	    REGION STATE MACHINE STEPS
	      CASE #statState OF
	        0://STATE 0
	          #statDriveControl.xDriveEnable := #statEnabled;
	          #statDriveControl.xDriveRun := FALSE;
	          #statDriveControl.xDriveEmergencyStop := #statSafetyIsOk;
	          #statDriveControl.iDriveSpeedRef_percent := 0.0;
	          #statBrushingIsDone := false;
	          #statBrushDriveControl.xDriveEnable := #statEnabled;
	          #statBrushDriveControl.xDriveRun := FALSE;
	          #statBrushDriveControl.xDriveEmergencyStop := #statSafetyIsOk;
	          #statBrushDriveControl.iDriveSpeedRef_percent := 0.0;
	          #statBrushing := false;
	          #statTrayStopperExtend := FALSE;
	          #statBrushingIsDoneLock := FALSE;

	        1://STATE 1
	          #statDriveControl.xDriveEnable := #statEnabled;
	          #statDriveControl.xDriveRun := TRUE;
	          #statDriveControl.xDriveEmergencyStop := #statSafetyIsOk;
	          #statDriveControl.iDriveSpeedRef_percent := #statSpeed_percent;
	          #statBrushing := FALSE;
	          #statBrushDriveControl.xDriveEnable := #statEnabled;
	          #statBrushDriveControl.xDriveEmergencyStop := #statSafetyIsOk;
	          #statBrushDriveControl.xDriveRun := FALSE;

	        2://STATE 2
	          #statDriveControl.xDriveEnable := #statEnabled;
	          #statDriveControl.xDriveRun := FALSE;
	          #statDriveControl.xDriveEmergencyStop := #statSafetyIsOk;
	          #statDriveControl.iDriveSpeedRef_percent := 0.0;
	          #statTrayStopperExtend := FALSE;
	        3://STATE 3
	          #statDriveControl.xDriveEnable := false;
	          #statDriveControl.xDriveRun := FALSE;
	          #statDriveControl.xDriveEmergencyStop := #statSafetyIsOk;
	          #statDriveControl.iDriveSpeedRef_percent := 0.0;
	          #statBrushing := FALSE;
	          #statTrayStopperExtend := FALSE;
	          #statBrushDriveControl.xDriveRun := FALSE;
	        4://STATE 4
	          #statDriveControl.xDriveEnable := #statEnabled;
	          #statDriveControl.xDriveRun := FALSE;
	          #statDriveControl.xDriveEmergencyStop := false;
	          #statDriveControl.iDriveSpeedRef_percent := 0.0;
	          #statBrushing := FALSE;
	          #statTrayStopperExtend := FALSE;
	          #statDriveControl.xDriveEmergencyStop := FALSE;
	        5://STATE 5
	          #statDriveControl.xDriveEnable := #statEnabled;
	          #statDriveControl.xDriveRun := FALSE;
	          #statDriveControl.xDriveEmergencyStop := #statSafetyIsOk;
	          #statDriveControl.iDriveSpeedRef_percent := 0.0;
	          #statBrushDriveControl.xDriveEnable := #statEnabled;
	          #statBrushDriveControl.xDriveRun := TRUE;
	          #statBrushDriveControl.xDriveEmergencyStop := #statSafetyIsOk;
	          #statBrushDriveControl.iDriveSpeedRef_percent := #ConveyorInterface.commands.rBrushSpeed_percent;
	          #statBrushing := TRUE;
	        6://STATE 6
	          #statDriveControl.xDriveEnable := #statEnabled;
	          #statDriveControl.xDriveRun := #statRunConvInMaintenance;
	          #statDriveControl.xDriveEmergencyStop := #statSafetyIsOk;
	          #statDriveControl.iDriveSpeedRef_percent := #statSpeedInMaintenance_percent;
	          #statBrushDriveControl.xDriveEnable := #statEnabled;
	          #statBrushDriveControl.xDriveRun := #statRunBrushInMaintenance;
	          #statBrushDriveControl.xDriveEmergencyStop := #statSafetyIsOk;
	          #statBrushDriveControl.iDriveSpeedRef_percent := #statBrushSpeed_percent;
	          #statBrushing := #statBrushExtendInMaintenance;
	          #statTrayStopperExtend := #statTrayStopperExtendInMaintenance;
	        ELSE
	          #statDriveControl.xDriveEnable := false;
	          #statDriveControl.xDriveRun := FALSE;
	          #statDriveControl.xDriveEmergencyStop := #statSafetyIsOk;
	          #statDriveControl.iDriveSpeedRef_percent := 0.0;
	          #statBrushing := false;
	          #statBrushDriveControl.xDriveEnable := false;
	          #statBrushDriveControl.xDriveRun := FALSE;
	          #statBrushDriveControl.xDriveEmergencyStop := #statSafetyIsOk;
	          #statBrushDriveControl.iDriveSpeedRef_percent := 0.0;

	      END_CASE;
	    END_REGION STATE MACHINE STEPS

	  END_REGION STATE MACHINE

	  REGION POST-STATE MACHINE OPERATIONS
	    //operations in this block will be implemented in each cycle, disregarding the state

	  END_REGION POST-STATE MACHINE OPERATONS

	END_REGION LOGIC

	REGION WRITE OUTPUTS, CALL SUBFUNCTIONS
	  //drive control
	  #instConveyorDrive(driveControl := #statDriveControl,
	                     inPI4 := #ConveyorInterface.inputs.i_ConveyorSEWdrivePI4,
	                     driveStatus => #statDriveStatus,
	                     outPO4 => #ConveyorInterface.outputs.q_ConveyorSEWdrivePO4);

	  #ConveyorInterface.status.xFault := #statDriveStatus.xDriveFault;
	  #ConveyorInterface.status.wFaultCode.%X0 := #statDriveStatus.xDriveFault;
	  #ConveyorInterface.status.iStatus := #statState;

	  //brush drive control
	  #instBrushDrive(driveControl:=#statBrushDriveControl,
	                  inPI4:=#ConveyorInterface.inputs.i_BrushDrivePI4,
	                  driveStatus=>#statBrushDriveStatus,
	                  outPO4=>#ConveyorInterface.outputs.q_BrushDrivePO4);

	  #ConveyorInterface.status.xFault := #ConveyorInterface.status.xFault OR #statBrushDriveStatus.xDriveFault;
	  #ConveyorInterface.status.wFaultCode.%X1 := #statBrushDriveStatus.xDriveFault;

	  //brush control
	  #ConveyorInterface.outputs.q_xBrushExtend := #statBrushing;
	  //stopper control
	  #ConveyorInterface.outputs.q_xTrayStopperExtend := #statTrayStopperExtend;

	END_REGION WRITE OUTPUTS, CALL SUBFUNCTIONS
END_FUNCTION_BLOCK

FUNCTION_BLOCK "ClassConveyorWithEjectSEW"
{ S7_Optimized_Access := 'TRUE' }
VERSION : 0.3
   VAR_IN_OUT
      ConveyorInterface : "typeConveyorWithEjectInterface";
   END_VAR

   VAR
      statEnabled { ExternalAccessible := 'False'; ExternalVisible := 'False'; ExternalWritable := 'False'} : Bool;
      instTimeDelay {InstructionName := 'TON_TIME'; LibVersion := '1.0'; ExternalAccessible := 'False'; ExternalVisible := 'False'; ExternalWritable := 'False'; S7_SetPoint := 'False'} : TON_TIME;
      statState { ExternalAccessible := 'False'; ExternalVisible := 'False'; ExternalWritable := 'False'} : USInt;   // State Machine Step number
      statNumberOfStates { ExternalAccessible := 'False'; ExternalVisible := 'False'; ExternalWritable := 'False'} : USInt := 1;   // State Machine Number of Steps
      statReadyForState { ExternalAccessible := 'False'; ExternalVisible := 'False'; ExternalWritable := 'False'} : Array[0..9] of Bool;
      statCycleCounter { ExternalAccessible := 'False'; ExternalVisible := 'False'; ExternalWritable := 'False'} : USInt;   // class specific variables
      statStart { ExternalAccessible := 'False'; ExternalVisible := 'False'; ExternalWritable := 'False'} : Bool;
      statStop { ExternalAccessible := 'False'; ExternalVisible := 'False'; ExternalWritable := 'False'} : Bool;
      statFull { ExternalAccessible := 'False'; ExternalVisible := 'False'; ExternalWritable := 'False'} : Bool;
      statSafetyIsOk { ExternalAccessible := 'False'; ExternalVisible := 'False'; ExternalWritable := 'False'} : Bool;
      statReset { ExternalAccessible := 'False'; ExternalVisible := 'False'; ExternalWritable := 'False'} : Bool;
      statMaintenance { ExternalAccessible := 'False'; ExternalVisible := 'False'; ExternalWritable := 'False'} : Bool;
      statRunConvInMaintenance { ExternalAccessible := 'False'; ExternalVisible := 'False'; ExternalWritable := 'False'} : Bool;
      statExtendEjectInMaintenance { ExternalAccessible := 'False'; ExternalVisible := 'False'; ExternalWritable := 'False'} : Bool;
      statSpeed_percent { ExternalAccessible := 'False'; ExternalVisible := 'False'; ExternalWritable := 'False'} : Real;
      statSpeedInMaintenance_percent { ExternalAccessible := 'False'; ExternalVisible := 'False'; ExternalWritable := 'False'} : Real;
      statStartOffTrigger { ExternalAccessible := 'False'; ExternalVisible := 'False'; ExternalWritable := 'False'} : Bool;
      statStopOnTrigger { ExternalAccessible := 'False'; ExternalVisible := 'False'; ExternalWritable := 'False'} : Bool;
      statFullOnTrigger { ExternalAccessible := 'False'; ExternalVisible := 'False'; ExternalWritable := 'False'} : Bool;
      statVFDfault { ExternalAccessible := 'False'; ExternalVisible := 'False'; ExternalWritable := 'False'} : Bool;
      statTrayEjected { ExternalAccessible := 'False'; ExternalVisible := 'False'; ExternalWritable := 'False'} : Bool;
      statDriveControl { ExternalAccessible := 'False'; ExternalVisible := 'False'; ExternalWritable := 'False'} : "typeDriveControl";
      statDriveStatus { ExternalAccessible := 'False'; ExternalVisible := 'False'; ExternalWritable := 'False'} : "typeDriveStatus";   // instances
      instConveyorStartOffDelay {InstructionName := 'TOF_TIME'; LibVersion := '1.0'; ExternalAccessible := 'False'; ExternalVisible := 'False'; ExternalWritable := 'False'; S7_SetPoint := 'False'} : TOF_TIME;
      instConveyorStopOnDelay {InstructionName := 'TON_TIME'; LibVersion := '1.0'; ExternalAccessible := 'False'; ExternalVisible := 'False'; ExternalWritable := 'False'; S7_SetPoint := 'False'} : TON_TIME;
      instConveyorFullOnDelay {InstructionName := 'TON_TIME'; LibVersion := '1.0'; ExternalAccessible := 'False'; ExternalVisible := 'False'; ExternalWritable := 'False'; S7_SetPoint := 'False'} : TON_TIME;
      instEjectDelay {InstructionName := 'TON_TIME'; LibVersion := '1.0'; ExternalAccessible := 'False'; ExternalVisible := 'False'; ExternalWritable := 'False'; S7_SetPoint := 'False'} : TON_TIME;
      instConveyorDrive { ExternalAccessible := 'False'; ExternalVisible := 'False'; ExternalWritable := 'False'; S7_SetPoint := 'False'} : "classDriveSEW";
   END_VAR

   VAR CONSTANT
      NUMBER_OF_STATES_IN_STATE_MACHINE : USInt := 7;   // 0-Conveyor stopped, 1-Conveyor running, 2-Conveyor full, 3-Conveyor fault, 4-Conveyor estopped, 5-Conveyor ejecting, 6-maintenance mode
   END_VAR


BEGIN
	REGION BLOCK INFO HEADER
	  //===============================================================================
	  // OTOMAKEIT SOLUTIONS / (c)Copyright 2024
	  //-------------------------------------------------------------------------------
	  // Title:            ClassConveyorWithEjectSEW
	  // Comment/Function: Conveyor class for TIA Portal, using SEW VFD drive. The only
	  //                   difference from the standard conveyor is the addition of the
	  //       eject cylinder control at the end of the conveyor
	  // Parental class:   classConveyor
	  // Library/Family:   LOMS (Library OtoMakeit Solutions)
	  // Author:           Yuriy Mosiyenko, Otomakeit Solutions
	  // Tested with:
	  // Engineering:      TIA Portal V17
	  // Restrictions:
	  // Requirements:     PLC (S7-1200 / S7-1500)
	  //-------------------------------------------------------------------------------
	  // Change log table:
	  //             | Date       | Expert in charge       | Changes applied
	  //-------------|------------|------------------------|------------------------------
	  // Created     | 2024-08-27 | Yuriy Mosiyenko        | Created
	  // Last update | 2024-08-29 | Yuriy Mosiyenko        | Corrections
	  //===============================================================================
	  //Update comments:
	  //-------------------------------------------------------------------------------
	  //2024-08-27 - Created the class
	  //2024-08-29 - Maintenance mode added
	  //===============================================================================
	  //===============================================================================
	END_REGION

	REGION INIT
	  #statNumberOfStates := #NUMBER_OF_STATES_IN_STATE_MACHINE;
	  FOR #statCycleCounter := 0 TO #statNumberOfStates DO
	    #statReadyForState[#statCycleCounter] := FALSE;
	  END_FOR;

	END_REGION INIT

	REGION READ INPUTS
	  #statEnabled := #ConveyorInterface.commands.xEnable;
	  #statStart := #ConveyorInterface.commands.xStart;
	  #statStop := #ConveyorInterface.commands.xStop;
	  #statFull := #ConveyorInterface.commands.xConveyorFullStatus;
	  #statReset := #ConveyorInterface.commands.xReset;
	  #statMaintenance := #ConveyorInterface.commands.xMaintenance;
	  #statRunConvInMaintenance := #ConveyorInterface.commands.xRunConvInMaintenance;
	  #statExtendEjectInMaintenance := #ConveyorInterface.commands.xExtendEjectInMaintenance;
	  #statSpeed_percent := #ConveyorInterface.commands.rConveyorSpeed_percent;
	  #statSpeedInMaintenance_percent := #ConveyorInterface.commands.rConveyorSpeedInMaintenance_percent;
	  #statSafetyIsOk := #ConveyorInterface.commands.xSafetyIsOk;

	END_REGION READ INPUTS

	REGION LOGIC

	  REGION PRE-STATE MACHINE OPERATIONS
	    //operations in this block will be implemented in each cycle, disregarding the state
	    //
	    //If reset received, reset faults, and set state machine to initial state
	    IF #statReset THEN
	      #ConveyorInterface.status.xFault := FALSE;
	      #ConveyorInterface.status.wFaultCode := 0;
	      #statState := 0;
	    END_IF;
	    IF NOT #statEnabled THEN //if the conveyor is disabled, stop it and set the status to 0 (stopped and ready)
	      #ConveyorInterface.status.iStatus := 0;
	      #statState := 0;
	      #statStart := FALSE;
	      #statStop := FALSE;
	    END_IF;
	    //start off delay
	    #instConveyorStartOffDelay(IN := #statStart,
	                               PT := #ConveyorInterface.commands.tStartOffDelay,
	                               Q => #statStartOffTrigger);
	    //STOP off delay
	    #instConveyorStopOnDelay(IN := #statStop,
	                              PT := #ConveyorInterface.commands.tStopOnDelay,
	                              Q => #statStopOnTrigger);
	    //FULL off delay
	    #instConveyorFullOnDelay(IN := #statFull,
	                              PT := #ConveyorInterface.commands.tFullOnDelay,
	                              Q => #statFullOnTrigger);
	    //Eject delay and output control
	    #instEjectDelay(IN := #statState = 5,
	                    PT := #ConveyorInterface.commands.tEjectTime,
	                    Q => #statTrayEjected);

	  END_REGION PRE-STATE MACHINE OPERATONS

	  REGION STATE MACHINE
	    REGION STATE MACHINE CONTROL
	      //set the conditions for each state
	      //state 0 - stopped and ready, state 1 - running, state 2 - stopped and full, state 3 - faulty, state 4 - estopped, state 5 - tray ejecting, state 6 - maintenance mode

	      //state 0 - if conveyor was full and the full status is removed or conveyor was running and the start or stop command is removed or fault was removed or safety was restored
	      //keep in mind that the stop command is active if false
	      #statReadyForState[0] := (#statState = 2 AND NOT #statFull)
	      OR (#statState = 4 AND #statSafetyIsOk)
	      OR (#statState = 3 AND NOT #statVFDfault)
	      OR (#statState = 5 AND #statTrayEjected)
	      OR (#statState = 6 AND NOT #statMaintenance);

	      //state 1 - if the conveyor is not full and the safety is ok and the start command is active
	      #statReadyForState[1] := (#statState = 0 AND #statStart AND #statSafetyIsOk);

	      //state 2 - if the conveyor is full
	      #statReadyForState[2] := (#statState < 3 AND #statFullOnTrigger AND #statSafetyIsOk);

	      //state 3 - if the VFD fault is detected
	      #statReadyForState[3] := (#statState = 1 AND #statVFDfault);

	      //state 4 - if the safety is not ok
	      #statReadyForState[4] := NOT #statSafetyIsOk;

	      //state 5 - if the stop command is active and delay is over
	      #statReadyForState[5] := (#statState = 1 AND #statStopOnTrigger AND #statSafetyIsOk);

	      //state 6 - if the maintenance mode is active
	      #statReadyForState[6] := (#statState = 0 AND #statMaintenance);

	      //change state if condition is TRUE
	      FOR #statCycleCounter := 0 TO #statNumberOfStates - 1 DO
	        IF #statReadyForState[#statCycleCounter] THEN
	          #statState := #statCycleCounter;
	        END_IF;
	      END_FOR;

	      //do not go over the set number of steps
	      IF #statState >= #statNumberOfStates THEN
	        #statState := 0;
	      END_IF;

	    END_REGION STATE MACHINE CONTROL

	    REGION STATE MACHINE STEPS
	      CASE #statState OF
	        0://STATE 0 - stopped and ready
	          #statDriveControl.xDriveEnable := #statEnabled;
	          #statDriveControl.xDriveRun := FALSE;
	          #statDriveControl.xDriveEmergencyStop := #statSafetyIsOk;
	          #statDriveControl.iDriveSpeedRef_percent := 0.0;
	          #statTrayEjected := FALSE;
	        1://STATE 1 - running
	          #statDriveControl.xDriveEnable := #statEnabled;
	          #statDriveControl.xDriveRun := TRUE;
	          #statDriveControl.xDriveEmergencyStop := #statSafetyIsOk;
	          #statDriveControl.iDriveSpeedRef_percent := #statSpeed_percent;
	        2://STATE 2 - stopped and full
	          #statDriveControl.xDriveEnable := #statEnabled;
	          #statDriveControl.xDriveRun := FALSE;
	          #statDriveControl.xDriveEmergencyStop := #statSafetyIsOk;
	          #statDriveControl.iDriveSpeedRef_percent := 0.0;
	        3://STATE 3 - faulty
	          #statDriveControl.xDriveEnable := false;
	          #statDriveControl.xDriveRun := FALSE;
	          #statDriveControl.xDriveEmergencyStop := #statSafetyIsOk;
	          #statDriveControl.iDriveSpeedRef_percent := 0.0;
	        4://STATE 4 - estopped
	          #statDriveControl.xDriveEnable := #statEnabled;
	          #statDriveControl.xDriveRun := FALSE;
	          #statDriveControl.xDriveEmergencyStop := false;
	          #statDriveControl.iDriveSpeedRef_percent := 0.0;
	        5://STATE 5 - tray ejecting
	          #statDriveControl.xDriveEnable := #statEnabled;
	          #statDriveControl.xDriveRun := FALSE;
	          #statDriveControl.xDriveEmergencyStop := #statSafetyIsOk;
	          #statDriveControl.iDriveSpeedRef_percent := 0.0;
	        6://STATE 6 - maintenance mode
	          #statDriveControl.xDriveEnable := #statEnabled;
	          #statDriveControl.xDriveRun := #statRunConvInMaintenance;
	          #statDriveControl.xDriveEmergencyStop := #statSafetyIsOk;
	          #statDriveControl.iDriveSpeedRef_percent := #statSpeedInMaintenance_percent;
	          #statExtendEjectInMaintenance := #statExtendEjectInMaintenance;

	        ELSE
	          #statDriveControl.xDriveEnable := false;
	          #statDriveControl.xDriveRun := FALSE;
	          #statDriveControl.xDriveEmergencyStop := #statSafetyIsOk;
	          #statDriveControl.iDriveSpeedRef_percent := 0.0;
	      END_CASE;
	    END_REGION STATE MACHINE STEPS

	  END_REGION STATE MACHINE

	  REGION POST-STATE MACHINE OPERATIONS
	    //operations in this block will be implemented in each cycle, disregarding the state

	  END_REGION POST-STATE MACHINE OPERATONS

	END_REGION LOGIC

	REGION WRITE OUTPUTS, CALL SUBFUNCTIONS
	  //drive control
	  #instConveyorDrive(driveControl := #statDriveControl,
	                     inPI4 := #ConveyorInterface.inputs.i_iConveyorSEWdrivePI4,
	                     driveStatus => #statDriveStatus,
	                     outPO4 => #ConveyorInterface.outputs.q_iConveyorSEWdrivePO4);

	  #ConveyorInterface.status.xFault := #statDriveStatus.xDriveFault;
	  #ConveyorInterface.status.wFaultCode := #statDriveStatus.wDriveFaultStatus;
	  #ConveyorInterface.status.iStatus := #statState;

	  //tray eject
	  IF #statState = 5 THEN
	    #ConveyorInterface.outputs.q_xTrayEject := TRUE;
	  ELSIF #statState = 6 THEN
	    #ConveyorInterface.outputs.q_xTrayEject := #statExtendEjectInMaintenance;
	  ELSE
	    #ConveyorInterface.outputs.q_xTrayEject := FALSE;
	  END_IF;

	END_REGION WRITE OUTPUTS, CALL SUBFUNCTIONS
END_FUNCTION_BLOCK

TYPE "typeOberlandTrayWashingLineInterface"
VERSION : 0.1
   STRUCT
      commands : Struct   // logical inputs to the block
         xEnable : Bool;
         xEstop : Bool;
         xFaultReset : Bool;
         xMaintenanceMode : Bool;
      END_STRUCT;
      status : Struct   // logical outputs from the block
         xFault : Bool;   // active fault on the line
         iState : USInt;   // status of the line, 0 - stopped and ready, 1 - running, 2 - faulty, 3 - estopped, 4 - maintenance mode
      END_STRUCT;
      inputs : Struct   // hardware inputs to the block   //Atomha interface inputs
         i_xAtomhaReadyToDeliverTray : Bool;
         i_xAtomhaReadyToReceiveTray : Bool;
      END_STRUCT;
      outputs : Struct   // hardware outputs from the blockAtomha interface outputs
         q_xABCOReadyToDeliverTray : Bool;
         q_xABCOReadyToReceiveTray : Bool;
      END_STRUCT;
      interfaces : Struct   // interfaces to the line
         io_InclineConveyorInterface : "typeConveyorInterface";
         io_PalletTipper01Interface : "typeConveyorTipperInterface";
         io_BrushConveyorInterface : "typeBrushingConveyorInterface";
         io_TakeAwayConveyorInterface : "typeConveyorWithEjectInterface";
         io_TransferConveyor01Interface : "typeConveyorInterface";
         io_InfeedAccumulationConveyorInterface : "typeConveyorInterface";
         io_InfeedConveyorInterface : "typeConveyorInterface";
         io_PalletWasherInterface : "typeConveyorPalletWasherSEW_Interface";
         io_PalletTipper02Interface : "typeConveyorTipperInterface";
         io_DischargeConveyorInterface : "typeConveyorWithEjectInterface";
         io_TransferConveyor02Interface : "typeConveyorInterface";
      END_STRUCT;
   END_STRUCT;

END_TYPE

FUNCTION_BLOCK "classOberlandTrayWashingLine"
{ S7_Optimized_Access := 'TRUE' }
VERSION : 0.2
   VAR_IN_OUT
      io_LineInterface : "typeOberlandTrayWashingLineInterface";   // State Machine variables
   END_VAR

   VAR
      statEstopTrigger { ExternalAccessible := 'False'; ExternalVisible := 'False'; ExternalWritable := 'False'} : Bool;
      statState { ExternalAccessible := 'False'; ExternalVisible := 'False'; ExternalWritable := 'False'} : USInt;   // State Machine Step number
      statNumberOfStates { ExternalAccessible := 'False'; ExternalVisible := 'False'; ExternalWritable := 'False'} : USInt := 1;   // State Machine Number of Steps
      statReadyForState { ExternalAccessible := 'False'; ExternalVisible := 'False'; ExternalWritable := 'False'} : Array[0..9] of Bool;
      statCycleCounter { ExternalAccessible := 'False'; ExternalVisible := 'False'; ExternalWritable := 'False'} : USInt;   // instance variablesinstance interfaces
      statInclineConveyorInterface { ExternalAccessible := 'False'; ExternalVisible := 'False'; ExternalWritable := 'False'} : "typeConveyorInterface";
      statPalletTipper01Interface { ExternalAccessible := 'False'; ExternalVisible := 'False'; ExternalWritable := 'False'} : "typeConveyorTipperInterface";
      statBrushConveyorInterface { ExternalAccessible := 'False'; ExternalVisible := 'False'; ExternalWritable := 'False'} : "typeBrushingConveyorInterface";
      statTakeAwayConveyorInterface { ExternalAccessible := 'False'; ExternalVisible := 'False'; ExternalWritable := 'False'} : "typeConveyorWithEjectInterface";
      statTransferConveyor01Interface { ExternalAccessible := 'False'; ExternalVisible := 'False'; ExternalWritable := 'False'} : "typeConveyorInterface";
      statInfeedAccumulationConveyorInterface { ExternalAccessible := 'False'; ExternalVisible := 'False'; ExternalWritable := 'False'} : "typeConveyorInterface";
      statInfeedConveyorInterface { ExternalAccessible := 'False'; ExternalVisible := 'False'; ExternalWritable := 'False'} : "typeConveyorInterface";
      statPalletWasherInterface { ExternalAccessible := 'False'; ExternalVisible := 'False'; ExternalWritable := 'False'} : "typeConveyorPalletWasherSEW_Interface";
      statPalletTipper02Interface { ExternalAccessible := 'False'; ExternalVisible := 'False'; ExternalWritable := 'False'} : "typeConveyorTipperInterface";
      statDischargeConveyorInterface { ExternalAccessible := 'False'; ExternalVisible := 'False'; ExternalWritable := 'False'} : "typeConveyorWithEjectInterface";
      statTransferConveyor02Interface { ExternalAccessible := 'False'; ExternalVisible := 'False'; ExternalWritable := 'False'} : "typeConveyorInterface";   // Instances of the line
      instInclineConveyor { ExternalAccessible := 'False'; ExternalVisible := 'False'; ExternalWritable := 'False'} : "ClassConveyorSEW";
      instPalletTipper01 { ExternalAccessible := 'False'; ExternalVisible := 'False'; ExternalWritable := 'False'} : "ClassConveyorTipperSEW";
      instBrushConveyor { ExternalAccessible := 'False'; ExternalVisible := 'False'; ExternalWritable := 'False'} : "ClassBrushingConveyorSEW";
      instTakeAwayConveyor { ExternalAccessible := 'False'; ExternalVisible := 'False'; ExternalWritable := 'False'} : "ClassConveyorWithEjectSEW";
      isntTransferConveyor01 { ExternalAccessible := 'False'; ExternalVisible := 'False'; ExternalWritable := 'False'} : "ClassConveyorSEW";
      instInfeedAccumulationConveyor { ExternalAccessible := 'False'; ExternalVisible := 'False'; ExternalWritable := 'False'} : "ClassConveyorSEW";
      instInfeedConveyor { ExternalAccessible := 'False'; ExternalVisible := 'False'; ExternalWritable := 'False'} : "ClassConveyorSEW";
      instPalletWasher { ExternalAccessible := 'False'; ExternalVisible := 'False'; ExternalWritable := 'False'} : "ClassConveyorPalletWasherSEW";
      instPalletTipper02 { ExternalAccessible := 'False'; ExternalVisible := 'False'; ExternalWritable := 'False'} : "ClassConveyorTipperSEW";
      instDischargeConveyor { ExternalAccessible := 'False'; ExternalVisible := 'False'; ExternalWritable := 'False'} : "ClassConveyorWithEjectSEW";
      instTransferConveyor02 { ExternalAccessible := 'False'; ExternalVisible := 'False'; ExternalWritable := 'False'} : "ClassConveyorSEW";
      instEstopDelay {InstructionName := 'TON_TIME'; LibVersion := '1.0'; ExternalAccessible := 'False'; ExternalVisible := 'False'; ExternalWritable := 'False'} : TON_TIME;
   END_VAR

   VAR CONSTANT
      NUMBER_OF_STATES_IN_STATE_MACHINE : USInt := 5;   // number of states in the state machine0 - stopped and ready, 1 - running, 2 - faulty, 3 - estopped, 4 - maintenance mode
   END_VAR


BEGIN
	REGION BLOCK INFO HEADER
	  //===============================================================================
	  // OTOMAKEIT SOLUTIONS / (c)Copyright 2024
	  //-------------------------------------------------------------------------------
	  // Title:            ABCO 32916 Washing Line Functions
	  // Comment/Function: System function block to control all the sequence flow of the
	  //                   line process
	  // Parental class:   LOMS_InOutTypeFB
	  //
	  // Library/Family:   LOMS (Library OtoMakeit Solutions)
	  // Author:           Yuriy Mosiyenko, Otomakeit Solutions
	  // Tested with:      CPU1215FC DC/DC/Relay
	  // Engineering:      TIA Portal V17
	  // Restrictions:
	  // Requirements:     PLC (S7-1200 / S7-1500)
	  //-------------------------------------------------------------------------------
	  // Change log table:
	  //             | Date       | Expert in charge       | Changes applied
	  //-------------|------------|------------------------|---------------------------
	  // Created     | 2024-08-28 | Yuriy Mosiyenko        | Created
	  // Last update | 2024-08-29 | Yuriy Mosiyenko        | Corrections
	  //===============================================================================
	  //Update comments:
	  //--------------------------------------------------------------------------------
	  //2024-08-28 - Created the class
	  //2024-08-29 - Added the maintenance mode
	  //================================================================================
	END_REGION

	REGION INIT
	  #statNumberOfStates := #NUMBER_OF_STATES_IN_STATE_MACHINE;
	  FOR #statCycleCounter := 0 TO #statNumberOfStates DO
	    #statReadyForState[#statCycleCounter] := FALSE;
	  END_FOR;

	  //reset fault status
	  #io_LineInterface.status.xFault := FALSE;

	  //E-Stop status delay timer (set to 10s for testing only!!!, make it not more than 1 sec after testing is done)
	  #instEstopDelay(IN := NOT #io_LineInterface.commands.xEstop,
	                  PT := T#10s,
	                  Q => #statEstopTrigger);

	END_REGION INIT

	REGION READ INTERFACES
	  //initially read all the interfaces from the Washing Line block interface
	  //and then assign different values only to the interface variables that are controlled by the block logic
	  #statInclineConveyorInterface.commands := #io_LineInterface.interfaces.io_InclineConveyorInterface.commands;
	  #statInclineConveyorInterface.inputs := #io_LineInterface.interfaces.io_InclineConveyorInterface.inputs;

	  #statPalletTipper01Interface.commands := #io_LineInterface.interfaces.io_PalletTipper01Interface.commands;
	  #statPalletTipper01Interface.inputs := #io_LineInterface.interfaces.io_PalletTipper01Interface.inputs;

	  #statBrushConveyorInterface.commands := #io_LineInterface.interfaces.io_BrushConveyorInterface.commands;
	  #statBrushConveyorInterface.inputs := #io_LineInterface.interfaces.io_BrushConveyorInterface.inputs;

	  #statTakeAwayConveyorInterface.commands := #io_LineInterface.interfaces.io_TakeAwayConveyorInterface.commands;
	  #statTakeAwayConveyorInterface.inputs := #io_LineInterface.interfaces.io_TakeAwayConveyorInterface.inputs;

	  #statTransferConveyor01Interface.commands := #io_LineInterface.interfaces.io_TransferConveyor01Interface.commands;
	  #statTransferConveyor01Interface.inputs := #io_LineInterface.interfaces.io_TransferConveyor01Interface.inputs;

	  #statInfeedAccumulationConveyorInterface.commands := #io_LineInterface.interfaces.io_InfeedAccumulationConveyorInterface.commands;
	  #statInfeedAccumulationConveyorInterface.inputs := #io_LineInterface.interfaces.io_InfeedAccumulationConveyorInterface.inputs;

	  #statInfeedConveyorInterface.commands := #io_LineInterface.interfaces.io_InfeedConveyorInterface.commands;
	  #statInfeedConveyorInterface.inputs := #io_LineInterface.interfaces.io_InfeedConveyorInterface.inputs;

	  #statPalletWasherInterface.commands := #io_LineInterface.interfaces.io_PalletWasherInterface.commands;
	  #statPalletWasherInterface.inputs := #io_LineInterface.interfaces.io_PalletWasherInterface.inputs;

	  #statPalletTipper02Interface.commands := #io_LineInterface.interfaces.io_PalletTipper02Interface.commands;
	  #statPalletWasherInterface.inputs := #io_LineInterface.interfaces.io_PalletWasherInterface.inputs;

	  #statDischargeConveyorInterface.commands := #io_LineInterface.interfaces.io_DischargeConveyorInterface.commands;
	  #statDischargeConveyorInterface.inputs := #io_LineInterface.interfaces.io_DischargeConveyorInterface.inputs;

	  #statTransferConveyor02Interface.commands := #io_LineInterface.interfaces.io_TransferConveyor02Interface.commands;
	  #statTransferConveyor02Interface.inputs := #io_LineInterface.interfaces.io_TransferConveyor02Interface.inputs;

	END_REGION READ INTERFACES

	REGION LOGIC

	  REGION PRE-STATE MACHINE OPERATIONS
	    //operations in this block will be implemented in each cycle, disregarding the state
	    //if the block is event-oriented, not sequence-oriented, put all the logic here. State
	    //machine block can be deleted in this case.

	  END_REGION PRE-STATE MACHINE OPERATONS

	  REGION STATE MACHINE
	    REGION STATE MACHINE CONTROL
	      //check conditions to change state
	      //replace FALSE with the condition
	      #statReadyForState[9] := FALSE;
	      #statReadyForState[8] := FALSE;
	      #statReadyForState[7] := FALSE;
	      #statReadyForState[6] := FALSE;
	      #statReadyForState[5] := FALSE;
	      //state 4 - maintenance mode
	      #statReadyForState[4] := #io_LineInterface.commands.xMaintenanceMode AND #statState = 0;
	      //state 3 - estopped
	      #statReadyForState[3] := NOT #io_LineInterface.commands.xEstop;
	      //state 2 - faulty
	      #statReadyForState[2] := #statState = 1 AND #io_LineInterface.status.xFault;
	      //state 1 - running
	      #statReadyForState[1] := #statState = 0 AND #io_LineInterface.commands.xEnable AND #io_LineInterface.commands.xEstop;
	      //state 0 - stopped and ready
	      #statReadyForState[0] := (#statState = 1 AND NOT #io_LineInterface.commands.xEnable)
	      OR (#statState = 2 AND #io_LineInterface.commands.xFaultReset AND NOT #io_LineInterface.status.xFault)
	      OR (#statState = 3 AND #io_LineInterface.commands.xEstop AND #io_LineInterface.commands.xFaultReset)
	      OR (#statState = 4 AND NOT #io_LineInterface.commands.xMaintenanceMode);

	      //change state if condition is TRUE
	      FOR #statCycleCounter := 0 TO #statNumberOfStates - 1 DO
	        IF #statReadyForState[#statCycleCounter] THEN
	          #statState := #statCycleCounter;
	        END_IF;
	      END_FOR;

	      //do not go over the set number of steps
	      IF #statState >= #statNumberOfStates THEN
	        #statState := 0;
	      END_IF;

	    END_REGION STATE MACHINE CONTROL

	    REGION STATE MACHINE STEPS
	      CASE #statState OF
	        0://STATE 0
	          //set the state of the line
	          #io_LineInterface.status.iState := 0;
	        1://STATE 1
	          //set the state of the line
	          #io_LineInterface.status.iState := 1;

	          //set the ready status to Atomha if there is no active full status
	          //on the Incline Conveyor
	          #io_LineInterface.outputs.q_xABCOReadyToReceiveTray := NOT #statInclineConveyorInterface.commands.xConveyorFullStatus;

	          //set the ready to deliver status to Atomha if there is a tray on the Transfer Conveyor 02 outfeed
	          #io_LineInterface.outputs.q_xABCOReadyToDeliverTray := #statTransferConveyor02Interface.commands.xStop;
	        2://STATE 2
	          //set the state of the line
	          #io_LineInterface.status.iState := 2;
	        3://STATE 3
	          //set the state of the line
	          #io_LineInterface.status.iState := 3;
	        4://STATE 4 - Maintenance Mode
	          //set the state of the line
	          #io_LineInterface.status.iState := 4;
	        ELSE
	          #statState := 0;
	      END_CASE;
	    END_REGION STATE MACHINE STEPS

	  END_REGION STATE MACHINE

	  REGION POST-STATE MACHINE OPERATIONS
	    //operations in this block will be implemented in each cycle, disregarding the state

	  END_REGION POST-STATE MACHINE OPERATONS

	END_REGION LOGIC

	REGION WRITE OUTPUTS, CALL SUBFUNCTIONS

	  REGION SUBFUNCTIONS
	    REGION Incline Conveyor
	      //set commands to the subfunction
	      //
	      #statInclineConveyorInterface.commands.xEnable := #io_LineInterface.commands.xEnable;
	      #statInclineConveyorInterface.commands.xSafetyIsOk := #io_LineInterface.commands.xEstop;
	      #statInclineConveyorInterface.commands.xReset := #io_LineInterface.commands.xFaultReset;
	      #statInclineConveyorInterface.commands.xMaintenance := #statState = 4;
	      #statInclineConveyorInterface.commands.rConveyorLength_cm := 563.88;
	      //start the conveyor only if Atomha is ready to deliver the tray
	      #statInclineConveyorInterface.commands.xStart := #statInclineConveyorInterface.commands.xStart
	      OR #io_LineInterface.inputs.i_xAtomhaReadyToDeliverTray;
	      //conveyor is full if both sensors are activated OR if the following tipper conveyor is busy with a tray
	      #statInclineConveyorInterface.commands.xConveyorFullStatus := #statInclineConveyorInterface.commands.xConveyorFullStatus
	      AND (#io_LineInterface.interfaces.io_PalletTipper01Interface.status.iStatus > 0);
	      //conveyor stop by the stop sensor only if the next conveyor is running yet
	      #statInclineConveyorInterface.commands.xStop := #statInclineConveyorInterface.commands.xStop
	      AND #io_LineInterface.interfaces.io_PalletTipper01Interface.status.iStatus > 0;
	      //call the subfunction
	      #instInclineConveyor(#statInclineConveyorInterface);
	      //collect all subfunction faults
	      #io_LineInterface.status.xFault := #io_LineInterface.status.xFault OR #statInclineConveyorInterface.status.xFault;
	      //outputs
	      #io_LineInterface.interfaces.io_InclineConveyorInterface.status := #statInclineConveyorInterface.status;
	      #io_LineInterface.interfaces.io_InclineConveyorInterface.outputs := #statInclineConveyorInterface.outputs;
	    END_REGION Incline Conveyor

	    REGION Pallet Tipper 01
	      //set commands to the subfunction
	      #statPalletTipper01Interface.commands.xEnable := #io_LineInterface.commands.xEnable;
	      #statPalletTipper01Interface.commands.xSafetyIsOk := #io_LineInterface.commands.xEstop;
	      #statPalletTipper01Interface.commands.xReset := #io_LineInterface.commands.xFaultReset;
	      #statPalletTipper01Interface.commands.xMaintenance := #statState = 4;
	      #statPalletTipper01Interface.commands.rConveyorLength_cm := 304.8;
	      //stop the conveyor only when the next conveyor is in running (not ready and standby)
	      #statPalletTipper01Interface.commands.xConveyorFullStatus := #statPalletTipper01Interface.commands.xConveyorFullStatus
	      OR #io_LineInterface.interfaces.io_BrushConveyorInterface.status.iStatus > 0;
	      //call the subfunction
	      #instPalletTipper01(#statPalletTipper01Interface);
	      //collect all subfunction faults
	      #io_LineInterface.status.xFault := #io_LineInterface.status.xFault OR #statPalletTipper01Interface.status.xFault;
	      //outputs
	      #io_LineInterface.interfaces.io_PalletTipper01Interface.status := #statPalletTipper01Interface.status;
	      #io_LineInterface.interfaces.io_PalletTipper01Interface.outputs := #statPalletTipper01Interface.outputs;
	    END_REGION Pallet Tipper 01

	    REGION Brush Conveyor
	      //set commands to the subfunction
	      #statBrushConveyorInterface.commands.xEnable := #io_LineInterface.commands.xEnable;
	      #statBrushConveyorInterface.commands.xSafetyIsOk := #io_LineInterface.commands.xEstop;
	      #statBrushConveyorInterface.commands.xReset := #io_LineInterface.commands.xFaultReset;
	      #statBrushConveyorInterface.commands.xMaintenance := #statState = 4;
	      #statBrushConveyorInterface.commands.rConveyorLength_cm := 393.7;
	      //call the subfunction
	      #instBrushConveyor(#statBrushConveyorInterface);
	      //collect all subfunction faults
	      #io_LineInterface.status.xFault := #io_LineInterface.status.xFault OR #statBrushConveyorInterface.status.xFault;
	      //outputs
	      #io_LineInterface.interfaces.io_BrushConveyorInterface.status := #statBrushConveyorInterface.status;
	      #io_LineInterface.interfaces.io_BrushConveyorInterface.outputs := #statBrushConveyorInterface.outputs;
	    END_REGION Brush Conveyor

	    REGION Take Away Conveyor
	      //set commands to the subfunction
	      #statTakeAwayConveyorInterface.commands.xEnable := #io_LineInterface.commands.xEnable;
	      #statTakeAwayConveyorInterface.commands.xSafetyIsOk := #io_LineInterface.commands.xEstop;
	      #statTakeAwayConveyorInterface.commands.xReset := #io_LineInterface.commands.xFaultReset;
	      #statTakeAwayConveyorInterface.commands.xMaintenance := #statState = 4;
	      #statTakeAwayConveyorInterface.commands.rConveyorLength_cm := 762.0;
	      //call the subfunction
	      #instTakeAwayConveyor(#statTakeAwayConveyorInterface);
	      //collect all subfunction faults
	      #io_LineInterface.status.xFault := #io_LineInterface.status.xFault OR #statTakeAwayConveyorInterface.status.xFault;
	      //outputs
	      #io_LineInterface.interfaces.io_TakeAwayConveyorInterface.status := #statTakeAwayConveyorInterface.status;
	      #io_LineInterface.interfaces.io_TakeAwayConveyorInterface.outputs := #statTakeAwayConveyorInterface.outputs;
	    END_REGION Take Away Conveyor

	    REGION Transfer Conveyor 01
	      //set commands to the subfunction
	      #statTransferConveyor01Interface.commands.xEnable := #io_LineInterface.commands.xEnable;
	      #statTransferConveyor01Interface.commands.xSafetyIsOk := #io_LineInterface.commands.xEstop;
	      #statTransferConveyor01Interface.commands.xReset := #io_LineInterface.commands.xFaultReset;
	      #statTransferConveyor01Interface.commands.xMaintenance := #statState = 4;
	      #statTransferConveyor01Interface.commands.rConveyorLength_cm := 246.38;
	      //signal transfer is full if washing conveyor is running
	      #statTransferConveyor01Interface.commands.xConveyorFullStatus := #io_LineInterface.interfaces.io_PalletWasherInterface.status.iConvStatus > 0;
	      //call the subfunction
	      #isntTransferConveyor01(#statTransferConveyor01Interface);
	      //collect all subfunction faults
	      #io_LineInterface.status.xFault := #io_LineInterface.status.xFault OR #statTransferConveyor01Interface.status.xFault;
	      //outputs
	      #io_LineInterface.interfaces.io_TransferConveyor01Interface.status := #statTransferConveyor01Interface.status;
	      #io_LineInterface.interfaces.io_TransferConveyor01Interface.outputs := #statTransferConveyor01Interface.outputs;
	    END_REGION Transfer Conveyor 01

	    REGION Infeed Accumulation Conveyor
	      //set commands to the subfunction
	      #statInfeedAccumulationConveyorInterface.commands.xEnable := #io_LineInterface.commands.xEnable;
	      #statInfeedAccumulationConveyorInterface.commands.xSafetyIsOk := #io_LineInterface.commands.xEstop;
	      #statInfeedAccumulationConveyorInterface.commands.xReset := #io_LineInterface.commands.xFaultReset;
	      #statInfeedAccumulationConveyorInterface.commands.xMaintenance := #statState = 4;
	      #statInfeedAccumulationConveyorInterface.commands.rConveyorLength_cm := 1178.56;
	      //signal infeed accum full if washing conveyor is running
	      #statInfeedAccumulationConveyorInterface.commands.xConveyorFullStatus := #io_LineInterface.interfaces.io_PalletWasherInterface.status.iConvStatus > 0;
	      //call the subfunction
	      #instInfeedAccumulationConveyor(#statInfeedAccumulationConveyorInterface);
	      //collect all subfunction faults
	      #io_LineInterface.status.xFault := #io_LineInterface.status.xFault OR #statInfeedAccumulationConveyorInterface.status.xFault;
	      //outputs
	      #io_LineInterface.interfaces.io_InfeedAccumulationConveyorInterface.status := #statInfeedAccumulationConveyorInterface.status;
	      #io_LineInterface.interfaces.io_InfeedAccumulationConveyorInterface.outputs := #statInfeedAccumulationConveyorInterface.outputs;
	    END_REGION Infeed Accumulation Conveyor

	    REGION Infeed Conveyor
	      //set commands to the subfunction
	      #statInfeedConveyorInterface.commands.xEnable := #io_LineInterface.commands.xEnable;
	      #statInfeedConveyorInterface.commands.xSafetyIsOk := #io_LineInterface.commands.xEstop;
	      #statInfeedConveyorInterface.commands.xReset := #io_LineInterface.commands.xFaultReset;
	      #statInfeedConveyorInterface.commands.xMaintenance := #statState = 4;
	      #statInfeedConveyorInterface.commands.rConveyorLength_cm := 152.4;
	      //call the subfunction
	      #instInfeedConveyor(#statInfeedConveyorInterface);
	      //collect all subfunction faults
	      #io_LineInterface.status.xFault := #io_LineInterface.status.xFault OR #statInfeedConveyorInterface.status.xFault;
	      //outputs
	      #io_LineInterface.interfaces.io_InfeedConveyorInterface.status := #statInfeedConveyorInterface.status;
	      #io_LineInterface.interfaces.io_InfeedConveyorInterface.outputs := #statInfeedConveyorInterface.outputs;
	    END_REGION Infeed Conveyor

	    REGION Pallet Washer
	      //set commands to the subfunction
	      #statPalletWasherInterface.commands.xEnable := #io_LineInterface.commands.xEnable;
	      #statPalletWasherInterface.commands.xSafetyIsOk := #io_LineInterface.commands.xEstop;
	      #statPalletWasherInterface.commands.xReset := #io_LineInterface.commands.xFaultReset;
	      #statPalletWasherInterface.commands.xMaintenance := #statState = 4;
	      #statPalletWasherInterface.commands.rConveyorLength_cm := 822.96;
	      //call the subfunction
	      #instPalletWasher(#statPalletWasherInterface);
	      //collect all subfunction faults
	      #io_LineInterface.status.xFault := #io_LineInterface.status.xFault OR #statPalletWasherInterface.status.xFault;
	      //outputs
	      #io_LineInterface.interfaces.io_PalletWasherInterface.status := #statPalletWasherInterface.status;
	      #io_LineInterface.interfaces.io_PalletWasherInterface.outputs := #statPalletWasherInterface.outputs;
	    END_REGION Pallet Washer

	    REGION Pallet Tipper 02
	      //set commands to the subfunction
	      #statPalletTipper02Interface.commands.xEnable := #io_LineInterface.commands.xEnable;
	      #statPalletTipper02Interface.commands.xSafetyIsOk := #io_LineInterface.commands.xEstop;
	      #statPalletTipper02Interface.commands.xReset := #io_LineInterface.commands.xFaultReset;
	      #statPalletTipper02Interface.commands.xMaintenance := #statState = 4;
	      #statPalletTipper02Interface.commands.rConveyorLength_cm := 304.8;
	      //call the subfunction
	      #instPalletTipper02(#statPalletTipper02Interface);
	      //collect all subfunction faults
	      #io_LineInterface.status.xFault := #io_LineInterface.status.xFault OR #statPalletTipper02Interface.status.xFault;
	      //outputs
	      #io_LineInterface.interfaces.io_PalletTipper02Interface.status := #statPalletTipper02Interface.status;
	      #io_LineInterface.interfaces.io_PalletTipper02Interface.outputs := #statPalletTipper02Interface.outputs;
	    END_REGION Pallet Tipper 02

	    REGION Discharge Conveyor
	      //set commands to the subfunction
	      #statDischargeConveyorInterface.commands.xEnable := #io_LineInterface.commands.xEnable;
	      #statDischargeConveyorInterface.commands.xSafetyIsOk := #io_LineInterface.commands.xEstop;
	      #statDischargeConveyorInterface.commands.xReset := #io_LineInterface.commands.xFaultReset;
	      #statDischargeConveyorInterface.commands.xMaintenance := #statState = 4;
	      #statDischargeConveyorInterface.commands.rConveyorLength_cm := 1016.0;
	      //call the subfunction
	      #instDischargeConveyor(#statDischargeConveyorInterface);
	      //collect all subfunction faults
	      #io_LineInterface.status.xFault := #io_LineInterface.status.xFault OR #statDischargeConveyorInterface.status.xFault;
	      //outputs
	      #io_LineInterface.interfaces.io_DischargeConveyorInterface.status := #statDischargeConveyorInterface.status;
	      #io_LineInterface.interfaces.io_DischargeConveyorInterface.outputs := #statDischargeConveyorInterface.outputs;
	    END_REGION Discharge Conveyor

	    REGION Transfer Conveyor 02
	      //set commands to the subfunction
	      #statTransferConveyor02Interface.commands.xEnable := #io_LineInterface.commands.xEnable;
	      #statTransferConveyor02Interface.commands.xSafetyIsOk := #io_LineInterface.commands.xEstop;
	      #statTransferConveyor02Interface.commands.xReset := #io_LineInterface.commands.xFaultReset;
	      #statTransferConveyor02Interface.commands.xMaintenance := #statState = 4;
	      #statTransferConveyor02Interface.commands.rConveyorLength_cm := 279.4;
	      //start the conveyor only if Atomha is ready to receive the tray
	      #statTransferConveyor02Interface.commands.xStart := #statTransferConveyor02Interface.commands.xStart AND #io_LineInterface.inputs.i_xAtomhaReadyToReceiveTray;
	      //call the subfunction
	      #instTransferConveyor02(#statTransferConveyor02Interface);
	      //collect all subfunction faults
	      #io_LineInterface.status.xFault := #io_LineInterface.status.xFault OR #statTransferConveyor02Interface.status.xFault;
	      //outputs
	      #io_LineInterface.interfaces.io_TransferConveyor02Interface.status := #statTransferConveyor02Interface.status;
	      #io_LineInterface.interfaces.io_TransferConveyor02Interface.outputs := #statTransferConveyor02Interface.outputs;
	    END_REGION Transfer Conveyor 02

	  END_REGION SUBFUNCTIONS

	END_REGION WRITE OUTPUTS, CALL SUBFUNCTIONS
END_FUNCTION_BLOCK

